TYPE MaxFilterPressure :
STRUCT
	LimitPressure: LREAL;
	OpenOnFilterAlarm: BOOL;
END_STRUCT
END_TYPE

(* stored: Version 1.1.0.1, ProductVersion 3.1.4024.6
   DUT MaxFilterPressure: Id {55e7756b-2383-4c6c-b3a9-4b74106b435f} *)
